# EPICS autosave request: leybold/read_int_floatE_settings.req
$(P):$(FPARAM)_RBV.HIGH
$(P):$(FPARAM)_RBV.HIHI
$(P):$(FPARAM)_RBV.LOLO
$(P):$(FPARAM)_RBV.LOW
